TYPE ST_AxisRecipe :
	STRUCT
		Velocity	 : LREAL := 100;
		Acceleration : LREAL := 1000;
		Deceleration : LREAL := 1000;
		Jerk		 : LREAL := 1000;
	END_STRUCT
END_TYPE

(* stored: Version 1.1.0.1
   DUT ST_AxisRecipe: Id {280e2d58-57ff-45cb-8736-8e6c02d6e056} *)
